Fanuc TP program (LS listing): template_2.ls

/PROG  TEMPLATE_2
/ATTR
OWNER		= MNEDITOR;
COMMENT		= "2"TEMPLATE SETUP";
PROG_SIZE	= 1023;
CREATE		= DATE 22-10-05  TIME 15:59:40;
MODIFIED	= DATE 23-09-29  TIME 17:30:04;
FILE_NAME	= ;
VERSION		= 0;
LINE_COUNT	= 44;
MEMORY_SIZE	= 1479;
PROTECT		= READ_WRITE;
TCD:  STACK_SIZE	= 0,
      TASK_PRIORITY	= 50,
      TIME_SLICE	= 0,
      BUSY_LAMP_OFF	= 0,
      ABORT_REQUEST	= 0,
      PAUSE_REQUEST	= 0;
DEFAULT_GROUP	= 1,*,*,*,*;
CONTROL_CODE	= 00000000 00000000;
/APPL
/APPL

AUTO_SINGULARITY_HEADER;
  ENABLE_SINGULARITY_AVOIDANCE   : TRUE;
/MN
   1:  --eg:SETUP FOR 2" TEMPLATE ;
   2:   ;
   3:  LBL[1:START] ;
   4:  --eg:SET TEMPLATE DIMENSIONS ;
   5:  R[1:ACTIVE TEMPLATE]=2    ;
   6:  R[10:NUMBER OF ROWS]=9    ;
   7:  R[11:NUMBER OF COLS]=23    ;
   8:  R[12:ROW SPACING (X)]=52    ;
   9:  R[13:COL SPACING (Y)]=45    ;
  10:  R[50:MIN DIAMETER]=12    ;
  11:  R[51:MAX DIAMETER]=53    ;
  12:  R[52:MIN LENGTH]=18    ;
  13:  R[53:MAX LENGTH]=280    ;
  14:   ;
  15:  --eg:USE LENGTH OF ONE SIDE OF TEMPLATE SQUARE. (A^2=B^2+C^2)/2 ;
  16:  R[84:SIDE LENGTH]=54.7878    ;
  17:  R[79:SLOT X CENTER]=38.62    ;
  18:   ;
  19:  LBL[2:SET SLOT USAGE] ;
  20:  --eg:SETS THE FIRST AND LAST COLUMN BEING USED IN EACH ROW AND WHICH
    :  SLOTS TO SKIP ;
  21:  R[14:ROW 1 START COL]=8    ;
  22:  R[15:ROW 1 STOP COL]=16    ;
  23:  R[16:ROW 2 START COL]=7    ;
  24:  R[17:ROW 2 STOP COL]=17    ;
  25:  R[18:ROW 3 START COL]=4    ;
  26:  R[19:ROW 3 STOP COL]=20    ;
  27:  R[20:ROW 4 START COL]=3    ;
  28:  R[21:ROW 4 STOP COL]=21    ;
  29:  R[22:ROW 5 START COL]=2    ;
  30:  R[23:ROW 5 STOP COL]=22    ;
  31:  R[24:ROW 6 START COL]=3    ;
  32:  R[25:ROW 6 STOP COL]=21    ;
  33:  R[26:ROW 7 START COL]=2    ;
  34:  R[27:ROW 7 STOP COL]=22    ;
  35:  R[28:ROW 8 START COL]=1    ;
  36:  R[29:ROW 8 STOP COL]=21    ;
  37:  R[30:ROW 9 START COL]=2    ;
  38:  R[31:ROW 9 STOP COL]=22    ;
  39:  R[32:1ST SLOT SKIP]=144    ;
  40:  R[33:2ND SLOT SKIP]=156    ;
  41:  R[34:3RD SLOT SKIP]=0    ;
  42:  R[35:4TH SLOT SKIP]=0    ;
  43:   ;
  44:  LBL[9999:END] ;
/POS
/END
